// TIA Portal V17 export
// export: Created 2024-01-30T08:49:13.7689557Z, ExportSetting WithDefaults, DisplayName Totally Integrated Automation Portal, DisplayVersion V17 Update 6, DisplayName TIA Portal Openness, DisplayVersion V17 Update 6, DisplayName TIA Portal Version Control Interface, DisplayVersion V17, DisplayName STEP 7 Professional, DisplayVersion V17 Update 6, DisplayName STEP 7 Safety, DisplayVersion V17 Update 6, DisplayName WinCC Advanced, DisplayVersion V17 Update 6
DATA_BLOCK "Gatewas_RS232_LK_G5000_DB"   // DB18
VERSION : 0.1
// stored: AutoNumber true, DBAccessibleFromOPCUA true, DBAccessibleFromWebserver true, InstanceOfName Gatewas_RS232_LK_G5000, InstanceOfType FB
"Gatewas_RS232_LK_G5000"
   // VAR_INPUT
   //    IN_COM : "UDT_LKG5000_RS232_RCV";
   //    IN_DATA : "UDT_RS232_RCV_DATA";
   //    SEND_TELEGRAM : Bool;
   //    COMMAND : String[10];
   // END_VAR
   // VAR_OUTPUT
   //    OUT_COM : "UDT_LKG5000_RS232_SEND";
   //    OUT_DATA : "UDT_RS232_SEND_DATA";
   // END_VAR
   // VAR
   //    COMMAND_SIGN : Array[0..10] of Char;
   //    Cnt_Command : UInt;
   //    IEC_Timer_0_Instance { S7_SetPoint := 'True'} : TOF_TIME;
   //    IEC_Timer_0_Instance_1 { S7_SetPoint := 'True'} : TOF_TIME;
   // END_VAR
BEGIN
END_DATA_BLOCK
